// TIA Portal project "Soru7" (V15)

(* hardware
DEVICE "S7-1200 station_1"  S7-1200 Station
   slot 0: "Rack_0"  S7-1200 Rack  Rack  V1.0
   slot 1: "PLC_1"  CPU 1214C DC/DC/DC  6ES7 214-1AG40-0XB0  V4.2
*)

// ===== PLC "PLC_1"  CPU 1214C DC/DC/DC =====

VAR_GLOBAL   // PLC tag table "Default tag table"
   "Duraklat_Baslat" AT %I0.0 : Bool;
   "Tag_1" AT %Q0.0 : Bool;
   "Oto için kırmızı" AT %Q0.1 : Bool;
   "oto için sarı" AT %Q0.2 : Bool;
   "oto için yeşil" AT %Q0.3 : Bool;
   "yaya için kırmızı" AT %Q0.4 : Bool;
   "yaya için yeşil" AT %Q0.5 : Bool;
   "Gece_Modu_mu" AT %I0.1 : Bool;
END_VAR

// folder: System blocks/Program resources

DATA_BLOCK "kirmizi_yesil_oto_yaya_H"   // DB1
{ S7_Optimized_Access := 'TRUE' }
AUTHOR : Simatic
FAMILY : IEC
NAME : IEC_TMR
VERSION : 1.0
// stored: InstanceOfName IEC_TIMER
"IEC_TIMER"
BEGIN
END_DATA_BLOCK

DATA_BLOCK "kirmizi_yesil_oto_yaya_L"   // DB2
{ S7_Optimized_Access := 'TRUE' }
AUTHOR : Simatic
FAMILY : IEC
NAME : IEC_TMR
VERSION : 1.0
// stored: InstanceOfName IEC_TIMER
"IEC_TIMER"
BEGIN
END_DATA_BLOCK

DATA_BLOCK "sari_L"   // DB3
{ S7_Optimized_Access := 'TRUE' }
AUTHOR : Simatic
FAMILY : IEC
NAME : IEC_TMR
VERSION : 1.0
// stored: InstanceOfName IEC_TIMER
"IEC_TIMER"
BEGIN
END_DATA_BLOCK

DATA_BLOCK "Sari_H"   // DB4
{ S7_Optimized_Access := 'TRUE' }
AUTHOR : Simatic
FAMILY : IEC
NAME : IEC_TMR
VERSION : 1.0
// stored: InstanceOfName IEC_TIMER
"IEC_TIMER"
BEGIN
END_DATA_BLOCK

DATA_BLOCK "gece_H"   // DB5
{ S7_Optimized_Access := 'TRUE' }
AUTHOR : Simatic
FAMILY : IEC
NAME : IEC_TMR
VERSION : 1.0
// stored: InstanceOfName IEC_TIMER
"IEC_TIMER"
BEGIN
END_DATA_BLOCK

DATA_BLOCK "Gece_L"   // DB6
{ S7_Optimized_Access := 'TRUE' }
AUTHOR : Simatic
FAMILY : IEC
NAME : IEC_TMR
VERSION : 1.0
// stored: InstanceOfName IEC_TIMER
"IEC_TIMER"
BEGIN
END_DATA_BLOCK

// folder: (top level)

ORGANIZATION_BLOCK "Main"   // OB1, LAD, ProgramCycle
TITLE = "Main Program Sweep (Cycle)"
{ S7_Optimized_Access := 'TRUE' }
VERSION : 0.1
   VAR_INPUT
      Initial_Call : Bool;   // Initial call of this OB
      Remanence : Bool;   // =True, if remanent data are available
   END_VAR
BEGIN

REGION Network 1: Otomabiler ve yaya için ortak olan kırmızı yeşil lamba zaman döngüleri
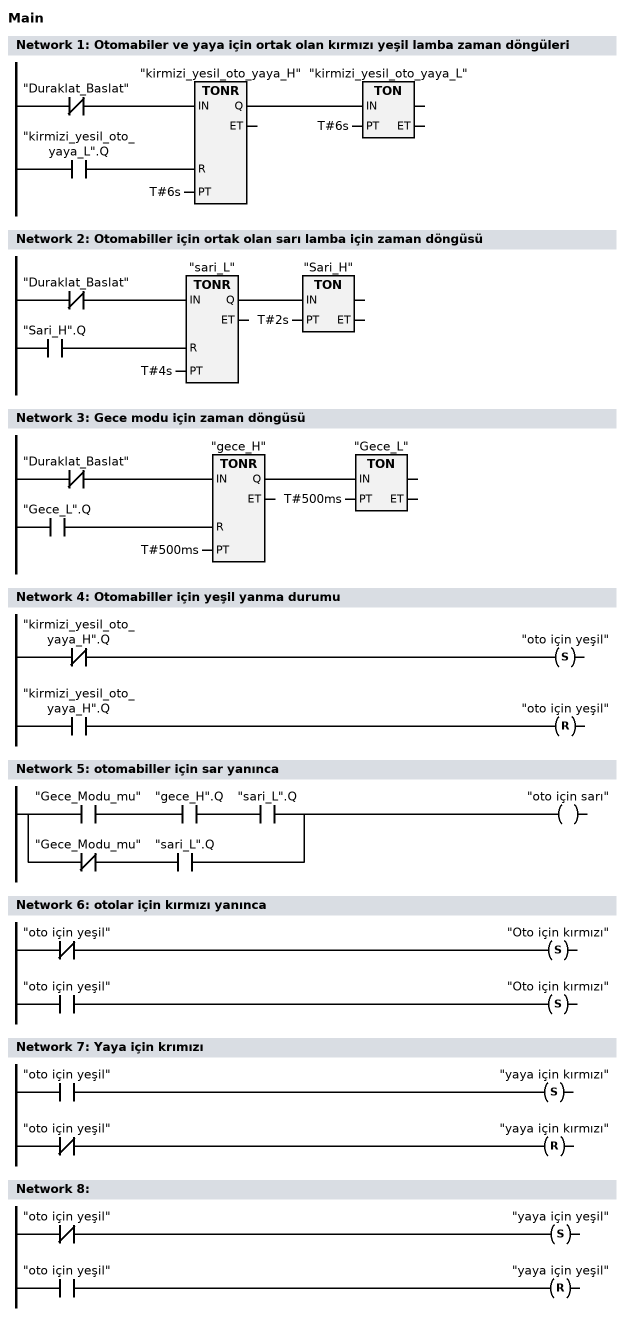
   "kirmizi_yesil_oto_yaya_H".TONR(IN := NOT "Duraklat_Baslat", R := "kirmizi_yesil_oto_yaya_L".Q, PT := T#6s);
   "kirmizi_yesil_oto_yaya_L".TON(IN := "kirmizi_yesil_oto_yaya_H".Q, PT := T#6s);
END_REGION

REGION Network 2: Otomabiller için ortak olan sarı lamba için zaman döngüsü
   "sari_L".TONR(IN := NOT "Duraklat_Baslat", R := "Sari_H".Q, PT := T#4s);
   "Sari_H".TON(IN := "sari_L".Q, PT := T#2s);
END_REGION

REGION Network 3: Gece modu için zaman döngüsü
   "gece_H".TONR(IN := NOT "Duraklat_Baslat", R := "Gece_L".Q, PT := T#500ms);
   "Gece_L".TON(IN := "gece_H".Q, PT := T#500ms);
END_REGION

REGION Network 4: Otomabiller için yeşil yanma durumu
   RUNG wire#powerrail
      I_Contact( "kirmizi_yesil_oto_yaya_H".Q )
      S_Coil( "oto için yeşil" )
   END_RUNG
   RUNG wire#powerrail
      Contact( "kirmizi_yesil_oto_yaya_H".Q )
      R_Coil( "oto için yeşil" )
   END_RUNG
   // the same network as SCL:
   IF NOT "kirmizi_yesil_oto_yaya_H".Q THEN "oto için yeşil" := TRUE; END_IF;
   IF "kirmizi_yesil_oto_yaya_H".Q THEN "oto için yeşil" := FALSE; END_IF;
END_REGION

REGION Network 5: otomabiller için sar yanınca
   RUNG wire#powerrail
      Contact( "Gece_Modu_mu" )
      Contact( "gece_H".Q )
      Contact( "sari_L".Q )
      wire#w1
      Coil( "oto için sarı" )
   END_RUNG
   RUNG wire#powerrail
      I_Contact( "Gece_Modu_mu" )
      Contact( "sari_L".Q )
   END_RUNG wire#w1
   // the same network as SCL:
   "oto için sarı" := ("Gece_Modu_mu" AND "gece_H".Q AND "sari_L".Q) OR (NOT "Gece_Modu_mu" AND "sari_L".Q);
END_REGION

REGION Network 6: otolar için kırmızı yanınca
   RUNG wire#powerrail
      I_Contact( "oto için yeşil" )
      S_Coil( "Oto için kırmızı" )
   END_RUNG
   RUNG wire#powerrail
      Contact( "oto için yeşil" )
      S_Coil( "Oto için kırmızı" )
   END_RUNG
   // the same network as SCL:
   IF NOT "oto için yeşil" THEN "Oto için kırmızı" := TRUE; END_IF;
   IF "oto için yeşil" THEN "Oto için kırmızı" := TRUE; END_IF;
END_REGION

REGION Network 7: Yaya için krımızı
   RUNG wire#powerrail
      Contact( "oto için yeşil" )
      S_Coil( "yaya için kırmızı" )
   END_RUNG
   RUNG wire#powerrail
      I_Contact( "oto için yeşil" )
      R_Coil( "yaya için kırmızı" )
   END_RUNG
   // the same network as SCL:
   IF "oto için yeşil" THEN "yaya için kırmızı" := TRUE; END_IF;
   IF NOT "oto için yeşil" THEN "yaya için kırmızı" := FALSE; END_IF;
END_REGION

REGION Network 8
   RUNG wire#powerrail
      I_Contact( "oto için yeşil" )
      S_Coil( "yaya için yeşil" )
   END_RUNG
   RUNG wire#powerrail
      Contact( "oto için yeşil" )
      R_Coil( "yaya için yeşil" )
   END_RUNG
   // the same network as SCL:
   IF NOT "oto için yeşil" THEN "yaya için yeşil" := TRUE; END_IF;
   IF "oto için yeşil" THEN "yaya için yeşil" := FALSE; END_IF;
END_REGION
END_ORGANIZATION_BLOCK